{attribute 'qualified_only'}
{attribute 'strict'}
TYPE E_Symo_PV_Error :
(
	eNoError := 0,
	eModbusTCPError := 1,
	eSymo10Error := 2,
	eSymo10TooBigValueReceived := 3
);
END_TYPE

(* stored: Version 1.1.0.1, ProductVersion 3.1.4024.9
   DUT E_Symo_PV_Error: Id {867d4510-bc80-4284-87c3-6b1ff591a0d3} *)
